RoboDK station: Raster Curve auto setup - Custom GUI.rdk

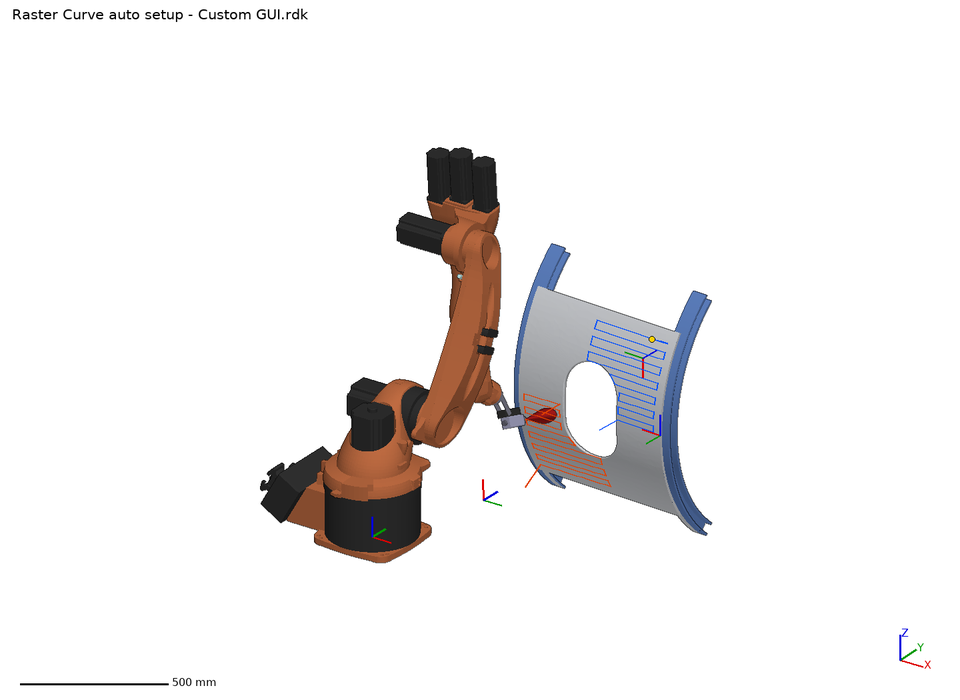
[picture v0: the station drawn from its stored meshes, robots at their saved joint values, targets as dots, program paths as lines]
Station Add curve sample project CreatePoint. Poses are relative to the parent item; angles as X-Y-Z fixed-axis rotations.
Station parameters (name, value as stored): IO_5, 0, CURVE_PARAMETERS, 600  600  250  250, STEP_X, 25.0, STEP_Y, 25.0, SPEED_OPERATION, 20.0, REPEAT_TIMES, 1.0, REPEAT_OFFSET, 2.0, ANGLE_TCP_X, 0.0, ANGLE_TCP_Y, -30.0, OVERTRAVEL, 25.0, SIZE_X, 300.0, SIZE_Y, 300.0
  - frame KUKA KR 5 arc Base at (0, 0, 0) mm
    - robot KUKA KR 5 arc: 6 axes, payload 5 kg, reach 1411 mm, repeatability 0.04 mm, weight 127 kg
        modified DH rows (alpha deg, a mm, theta deg, d mm): 0, 0, 0, 400; -90, 180, 0, 0; 0, 600, -90, 0; -90, 120, 0, 620; 90, 0, 0, 0; -90, 0, 180, 115
        joint limits [-155, -180, -15, -350, -130, -350] to [155, 65, 158, 350, 130, 350]; home [0, -90, 90, 0, 0, 0]; saved at [-90.662, -65.515, 150.914, 153.218, 47.362, 35.247]
      - tool Paint gun, TCP at (25, 0, 225) mm, rotated rx 0 ry 30 rz 0 deg, size 101.6 x 139.9 x 235.8 mm
    - frame CAD reference at (526.25, 941.36, 152.38) mm, rotated rx 0 ry 0 rz 177.82 deg
      - object Inspection Part at (0, 0, 0) mm, size 656 x 251.4 x 904.5 mm, 19 curves, geometry from Do something->PointOperations DOSOMETHING %ID%
      - frame Section1 at (31.6, 54.02, 303.28) mm, rotated rx 0 ry 90 rz -90 deg
        - object Section1 at (0, 0, 0) mm
      - frame Section2 at (569.12, 235.23, -318.39) mm, rotated rx 41.21 ry -87.7 rz 48.72 deg
        - object Section2 at (0, 0, 0) mm
  - Python program PointOperations (listed below)
  - Python program Curve_Auto_Setup (listed below)
  - machining project Section1: rotZ(0) | rotz(0) | onStart | onPathStart | onApproach | onPoint | onRetract | onFinish | Extruder(%1) | default | default | OutOnMov(%1) | OutOffMov(%1) | onPathFinish
  - program Section1 (141 instructions, listed below)
  - machining project Section2: rotZ(0) | onStart | onPathStart | onApproach | onPoint | onRetract | onFinish | Extruder(%1) | default | default | OutOnMov(%1) | OutOffMov(%1) | onPathFinish
  - program Section2 (141 instructions, listed below)
  - program MainInspection Part (2 instructions, listed below)
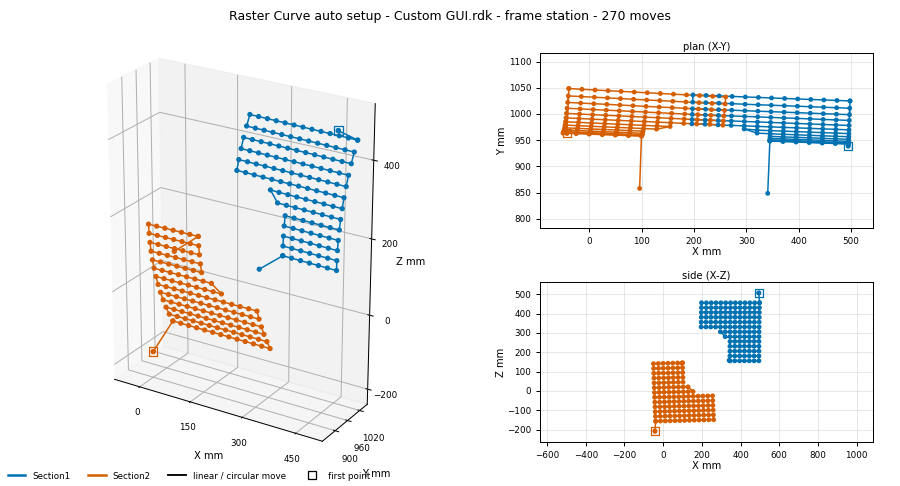
[picture p0: tool path of Raster Curve auto setup - Custom GUI.rdk in frame station, 270 of 270 moves have a stored position in this frame; points joined in program order, loops and branches not executed]

--- Python program PointOperations ---
import sys                # allows getting the argument parameters
from robodk import *      # required by mbox()
from robolink import *    # API to communicate with RoboDK

print('Number of arguments: ' + str(len(sys.argv)) + ' arguments.')

OBJECT = None
COMMAND = "SHOWPOINT_ALL"  # set to: NEWPOINT, SHOWPOINT

RDK = Robolink()

if len(sys.argv) >= 3:
    COMMAND = sys.argv[1]
    OBJECT = Item(RDK, int(sys.argv[2]))
    #RDK.ShowMessage("%s : %s" % (str(sys.argv), COMMAND))

else:
    OBJECT = RDK.ItemUserPick("Select an object", ITEM_TYPE_OBJECT)
    if not OBJECT.Valid():
        quit()

print("Selected object: %s" % OBJECT.Name())

if COMMAND == "SHOWPOINT_ALL":
    # Show all points in the object
    points, name = OBJECT.GetPoints(FEATURE_POINT)
    message = 'List of points for object<br>%s<br>' % OBJECT.Name()
    i = 0
    for pt in points:
        i = i + 1
        message += "p%i : %.3f , %.3f , %.3f <br>" % (i, pt[0], pt[1], pt[2])

    RDK.ShowMessage(message)

elif COMMAND == "SHOWPOINT":
    # Shows the point selected
    is_selected, feature_type, feature_id = OBJECT.SelectedFeature()
    points, name_selected = OBJECT.GetPoints(feature_type, feature_id)
    point = None
    if len(points) > 1:
        point = points[feature_id]
    else:
        point = points[0]
    RDK.ShowMessage("Selected Point: %s<br>XYZ = [%.3f, %.3f, %.3f]<br>ijk = [%.3f, %.3f, %.3f]" % (name_selected, point[0], point[1], point[2], point[3], point[4], point[5]))

elif COMMAND == "NEWPOINT":
    # create a new point under the mouse cursor
    point_mouse, name_feature = OBJECT.GetPoints(FEATURE_SURFACE)
    if 'point on surface' in name_feature.lower():
        point_rel = point_mouse[0]
        RDK.ShowMessage("%s -> XYZ = [%.3f, %.3f, %.3f] , ijk = [%.3f, %.3f, %.3f]" % (name_feature, point_rel[0], point_rel[1], point_rel[2], point_rel[3], point_rel[4], point_rel[5]), False)
        ADD_POINT_ON_OBJECT = True
        OBJECT.AddPoints([point_rel], ADD_POINT_ON_OBJECT, PROJECTION_NONE)
    else:
        RDK.ShowMessage("Select a surface")
else:
    raise Exception("Invalid operation specified")

--- Python program Curve_Auto_Setup ---
# Press F5 to run the script
# Type help("robolink") or help("robodk") for more information
#
# This script shows an example to create a raster curve that can be added programmatically to a RoboDK station
# The curve can be optionally projected to an existing object (either along the curve normals or a projection the closest surface)
#
# projection types (for AddCurve, as defined in robolink.py):
#PROJECTION_NONE                = 0 # No curve projection
#PROJECTION_CLOSEST             = 1 # The projection will the closest point on the surface
#PROJECTION_ALONG_NORMAL        = 2 # The projection will be done along the normal.
#PROJECTION_ALONG_NORMAL_RECALC = 3 # The projection will be done along the normal. Furthermore, the normal will be recalculated according to the surface normal.
#
# More information about the RoboDK API here:
# https://robodk.com/doc/en/PythonAPI/robolink.html
# https://robodk.com/doc/en/RoboDK-API.html
#
# This macro involves advanced Python programming as it uses the exec() and eval() statements to execute Python code from a string generated on the fly.
# The GUI is created automatically based on the variables defined in PARAM_VARS (global variables) and PARAM_LABELS (description to show on the menu)


# Set default/global parameters. This is only useful for the first time we execute this macro on a new RDK file.
# These global parameters are saved with the RoboDK station as Station parameters (right click the Station root and select "Station Parameters" to see the parameters saved)
SIZE_X = 500   # Size along the X axis
SIZE_Y = 500   # Size along the Y axis
STEP_X = 20    # Step along the X axis
STEP_Y = 50    # Step along the Y axis
SPEED_OPERATION = 20 # Operation speed
REPEAT_TIMES = 3    # Number of times to run the same program
REPEAT_OFFSET = 2   # Offset along Z axis in mm
ANGLE_TCP_X = 10
ANGLE_TCP_Y = 20
OVERTRAVEL = 25

REMEMBER_LAST_VALUES = True

#--------------------------------------------
# List the variables that will be remembered by the station and provided through the GUI
PARAM_VARS = []
PARAM_LABELS = []
PARAM_VARS += ["STEP_X", "STEP_Y"]
PARAM_LABELS += ["Step along X (mm)", "Step along Y (mm)"]

PARAM_VARS += ["SPEED_OPERATION"]
PARAM_LABELS +=  ["Operation speed (mm/s)"]

PARAM_VARS += ["REPEAT_TIMES", "REPEAT_OFFSET"]
PARAM_LABELS +=  ["Repeat times", "Repeat Offset along Z (mm)"]

PARAM_VARS += ["ANGLE_TCP_X", "ANGLE_TCP_Y"]
PARAM_LABELS +=  ["Tool angle X (deg)", "Tool angle Y (deg)"]

PARAM_VARS += ["OVERTRAVEL"]
PARAM_LABELS +=  ["Overtravel (mm)"]

PARAM_VARS += ["SIZE_X", "SIZE_Y"]
PARAM_LABELS += ["Size along X (mm)", "Size along Y (mm)"]

# Optionally provide a part name to auto select it without asking the user
PART_NAME = None # 'Paint Part'

#------------------------------------------------------------------
#--------------- PROGRAM START ---------------------
from robolink import *    # API to communicate with RoboDK
from robodk import *      # basic matrix operations

# Initialize the RoboDK API
RDK = Robolink()

# Set other constants:
TOL_PROJ_Z = sqrt(2)    # Tolerance to ignore a point as a ratio (if it falls through a window for example)

#---------------------------------------------
# First: Retrieve the part item
# Name of the reference used for the path projection
#

if PART_NAME is None:
    PART = RDK.ItemUserPick("Select a part", ITEM_TYPE_OBJECT)
    if PART is None:
        print("Operation cancelled by user")
        quit()
else:
    PART = RDK.Item(PART_NAME, ITEM_TYPE_OBJECT)

if not PART.Valid():
    raise Exception("The selected part is not valid or not available")

#---------------------------------------------
# List all the reference frames that we want to use to create
# raster paths (references attached to the object reference
part_ref = PART.Parent()

# Get the list of items attached to the part reference
ref_pattern_candidates = part_ref.Childs()
# Iterate through these child items and list the reference frames
# optionally add ignore in the name
REF_PATTERN_LIST = []
for ref_i in ref_pattern_candidates:
    if ref_i.Type() == ITEM_TYPE_FRAME and (not "ignore" in ref_i.Name()):
        REF_PATTERN_LIST.append(ref_i)

if len(REF_PATTERN_LIST) <= 0:
    RDK.ShowMessage("No reference frames found. Add one or more frames to " + part_ref.Name())
    quit()

#---------------------------------------------
# Retrieve Global parameters or set defaults as found in RoboDK
if REMEMBER_LAST_VALUES:
    for strvar in PARAM_VARS:
        var_value = RDK.getParam(strvar)
        if var_value is not None:
            exec(strvar + " = " + str(var_value))

#---------------------------------------------
# Load GUI tools
from tkinter import *
import tkinter.font as font

# Generate the main window
root = Tk()
root.title("Toolpath parameters")

# define a label to notify the user
NotifyGUI = StringVar()

#---------------------------------------------
# Function to change the coordinates of a point and a normal
# given a pose. The point and the normal must be in xyzijk format
def Pose_x_XYZijk(pose, xyzijk):
    new_xyz = pose*xyzijk[0:3]
    new_ijk = pose[:3,:3]*xyzijk[3:6]
    return new_xyz + new_ijk

#---------------------------------------------
# Function definition to create a list of points as zig-zag pattern (curve)
def GridPoints(ref, size_x, size_y, step_x, step_y):
    """Generates a list of points given dimensions of a grid"""
    points = []
    xx = 0
    flip = 1
    while xx <= size_x:
        yy = 0
        if flip > 0:
            yy = 0
        else:
            yy = size_y

        while yy <= size_y and yy >= 0:
            # Create a new point as [x,y,z , i,j,k]
            xyzijk = Pose_x_XYZijk(ref, [xx,yy,0 , 0,0,-1])
            points.append(xyzijk)
            yy = yy + flip*step_y

        xx = xx + step_x
        flip = -1*flip
    return points

#---------------------------------------------
# Function definition to offset a list of points
def PointsOffset(points, offset):
    points_offset = []
    for pi in points:
        x,y,z,i,j,k = pi
        xyz2 = add3([x,y,z], mult3([i,j,k], offset))
        xyzijk2 = xyz2 + [i,j,k]
        points_offset.append(xyzijk2)
    return points_offset

# Show message through the GUI, RoboDK and the console
def ShowMsg(msg):
    print(msg)
    NotifyGUI.set(msg)
    root.update_idletasks()
    RDK.ShowMessage(msg, False)

#---------------------------------------------
# Main program call that will project the path to a surface
def CreatePaths():
    prog_name_list = []
    for REF in REF_PATTERN_LIST:
        # Retrieve the reference name
        REF_NAME = REF.Name()

        ShowMsg("Working with %s ..." % REF_NAME)

        # Get the pose of the reference with respect to the part:
        pose_ref_wrt_part = invH(PART.Parent().PoseAbs())*REF.PoseAbs()

        # For later: calculate the inverse pose (part with respect to the reference)
        pose_part_wrt_ref = invH(pose_ref_wrt_part)

        # Generate the curve path
        # IMPORTANT: the point coordinates must be relative to the part reference
        points = GridPoints(pose_ref_wrt_part, SIZE_X, SIZE_Y, STEP_X, STEP_Y)
        # points is a list of points with respect to the part
        # Another option is to load the grid from a CSV file:
        #file = RDK.getParam('PATH_OPENSTATION') + '/test.csv'
        #POINTS = LoadList(file)
        #POINTS.pop(0)
        # display the points
        #print(CURVE)
        if len(points) == 0:
            ShowMsg("No points found for: " + REF_NAME)
            continue

        # Project the points on the object surface
        #pts_projected = PART.AddPoints(POINTS)
        ShowMsg("Projecting %s to surface..." % REF_NAME)
        points_projected = PART.ProjectPoints(Mat(points).tr(), PROJECTION_ALONG_NORMAL_RECALC)

        # Patch
        points_projected = points_projected.tr().rows

        points_projected_filtered = []

        ShowMsg("Filtering %s..." % REF_NAME)

        # Remember the last valid projection
        pti_last = None
        for i in range(0,len(points_projected)-1):
            # retrieve projected and non projected points, with respect to the reference frame
            # retrieve the next point to test if the projection went too far
            pti = Pose_x_XYZijk(pose_part_wrt_ref, points[i])
            pti_proj = Pose_x_XYZijk(pose_part_wrt_ref, points_projected[i])

            # Ignore non projected points (z coordinate is 0 mm, prevent numerical errors as well)
            if abs(pti_proj[2]) < 0.1:
                continue

            # Check if we have the first valid projected point
            if pti_last is None:
                points_projected_filtered.append(pti_proj)
                pti_last = pti
                pti_proj_last = pti_proj
                continue

            # Check if the projection falls through a "window" or "climbs" a wall with respect to the previous pointS
            if distance(pti_proj, pti_proj_last) < TOL_PROJ_Z*distance(pti, pti_last):
                # List the point as valid
                points_projected_filtered.append(pti_proj)

                # Remember the last valid projection
                pti_last = pti
                pti_proj_last = pti_proj

        # Remove any previously generated objects with the same name as the reference frame:
        obj_delete = RDK.Item(REF_NAME, ITEM_TYPE_OBJECT)
        if obj_delete.Valid():
            obj_delete.Delete()

        ShowMsg("Creating object for %s..." % REF_NAME)
        # Add the points as an object in the RoboDK station tree
        points_object = RDK.AddCurve(points_projected_filtered)
        # Add the points to the reference and set the reference name
        points_object.setParent(REF)
        points_object.setName(REF_NAME)

        for rep in range(1,round(REPEAT_TIMES)):
            # Calculate a new curve with respect to the reference curve
            points_projected_filtered_rep = PointsOffset(points_projected_filtered, REPEAT_OFFSET * rep)

            #  Add the shifted curve without projecting it
            points_object = RDK.AddCurve(points_projected_filtered_rep, points_object, True, PROJECTION_NONE)


        curve_follow = RDK.Item(REF_NAME, ITEM_TYPE_MACHINING)
        if not curve_follow.Valid():
            curve_follow = RDK.AddMillingProject(REF_NAME)

        ShowMsg("Solving toolpath for %s" % REF_NAME)

        # Use the current reference frame:
        curve_follow.setPoseFrame(REF)

        # RoboDK 3.3.7 or later required:
        curve_follow.setSpeed(SPEED_OPERATION)
        curve_follow.setPoseTool(rotx(ANGLE_TCP_X*pi/180.0)*roty(ANGLE_TCP_Y*pi/180.0))
        prog, status = curve_follow.setMillingParameters(part=points_object)
        print(status)
        if status == 0:
            ShowMsg("Program %s generated successfully" % REF_NAME)
        else:
            ShowMsg("Issues found generating program %s!" % REF_NAME)


        # get the program name
        prog_name = prog.Name()
        prog_name_list.append(prog_name)

    # Create a new program that calls the auto generated program
    # Make sure we delete any previously generated programs with the same name
    ShowMsg("Creating Main program ...")
    prog_main_name = "Main" + PART.Name()
    prog_main = RDK.Item(prog_main_name, ITEM_TYPE_PROGRAM)
    if prog_main.Valid():
        prog_main.Delete()
    prog_main = RDK.AddProgram(prog_main_name)

    # Add a number of program calls to the first program by providing inline code
    #prog_main.RunCodeCustom("FOR i=1 TO 5", INSTRUCTION_INSERT_CODE)
    #prog_main.RunCodeCustom(prog_name, INSTRUCTION_CALL_PROGRAM)
    #prog_main.RunCodeCustom("NEXT", INSTRUCTION_INSERT_CODE)
    #for i in range(4):
    for pr_name in prog_name_list:
        prog_main.RunCodeCustom(pr_name, INSTRUCTION_CALL_PROGRAM)


    # Start the program simulation:
    prog_main.RunProgram()
    ShowMsg("Done!!")


#-----------------------------------------
# Create a GUI menu using tkinter



# Use StringVar variables linked to the global variables for the GUI
txtSpeed_Operation = StringVar()
txtSpeed_Operation.set(str(SPEED_OPERATION))


for strvar, hint in zip(PARAM_VARS, PARAM_LABELS):
    var = eval(strvar)
    txtvar = "txt" + strvar
    #txtSize_X = StringVar()
    #txtSize_X.set(str(SIZE_X))
    #Label(root, text="Window Size X (mm)").pack()
    #Entry(root, textvariable=txtSize_X).pack()
    exec(txtvar + " = StringVar()")
    exec(txtvar + ".set(str(" + str(var) + "))")
    exec("Label(root, text='" + hint + "').pack()")
    exec("Entry(root, textvariable=" + txtvar + ").pack()")


# Add a button and default action to execute the current choice of the user
def btnUpdate():
    # List the global variables so that we can read or modify the latest values
    #exec(PARAM_GLOBALS)

    try:
        for strvar in PARAM_VARS:
            #SIZE_X = float(txtSize_X.get())
            # Update global variable
            exec("%s = float(txt%s.get())" % (strvar, strvar), globals())

    except Exception as e:
        RDK.ShowMessage("Invalid input!! " + str(e), False)
        return

    # Remember the last settings in the RoboDK station
    for strvar in PARAM_VARS:
        value = eval(strvar)
        RDK.setParam(strvar, value)

    # Run the main program once all the global variables have been set
    CreatePaths()

# Add an update button that calls btnUpdate()
font_large = font.Font(family='Helvetica', size=18, weight=font.BOLD)
Label(root, text=" ").pack() # Just a spacer
Label(root, textvariable=NotifyGUI).pack() # information variable
Button(root, text='Update', font=font_large, width=20, height=4, command=btnUpdate, bg='green').pack()

# Important to display the graphical user interface
root.mainloop()

--- program Section1 (robot KUKA KR 5 arc) ---
  Set Ref.: Section1
  Set Tool: Paint gun
  Show Paint gun
  Set speed (1000.0 mm/s)
  MoveJ 1 to (-50.79, 0.22, 50.26) mm, rotated rx 34.39 ry 25.95 rz 105.39 deg; joints [-51.825, -81.117, 121.806, -97.903, 30.623, 30.499]
  MoveL 2 to (-50.79, 0.22, 50.26) mm, rotated rx 34.39 ry 25.95 rz 105.39 deg; joints [-51.825, -81.117, 121.806, -97.903, 30.623, 30.499]
  MoveL 3 to (0, 0, 136.4) mm, rotated rx 34.39 ry 25.95 rz 105.39 deg; joints [-55.067, -72.344, 116.19, -106.364, 28.938, 37.73]
  MoveL 4 to (0, 0, 136.4) mm, rotated rx 34.39 ry 25.95 rz 105.39 deg; joints [-55.067, -72.344, 116.19, -106.364, 28.938, 37.73]
  Set speed (20.0 mm/s)
  MoveL 5 to (0, 25, 136.39) mm, rotated rx 34.36 ry 26.11 rz 105.47 deg; joints [-56.374, -73.392, 117.629, -108.355, 28.338, 38.991]
  MoveL 6 to (0, 50, 136.37) mm, rotated rx 34.57 ry 26.16 rz 105.61 deg; joints [-57.765, -74.441, 118.921, -109.961, 27.461, 39.815]
  MoveL 7 to (0, 75, 136.32) mm, rotated rx 34.08 ry 26.14 rz 105.33 deg; joints [-59.224, -75.485, 120.503, -113.62, 26.851, 42.548]
  MoveL 8 to (0, 100, 136.36) mm, rotated rx 35.34 ry 25.72 rz 105.77 deg; joints [-60.883, -76.578, 121.224, -113.176, 24.731, 41.191]
  MoveL 9 to (0, 125, 136.35) mm, rotated rx 34.79 ry 26.08 rz 105.68 deg; joints [-62.268, -77.415, 122.604, -116.74, 24.649, 43.9]
  MoveL 10 to (0, 150, 136.37) mm, rotated rx 33.98 ry 26.51 rz 105.48 deg; joints [-63.673, -78.184, 124.024, -120.948, 24.856, 47.226]
  MoveL 11 to (0, 175, 136.42) mm, rotated rx 34.8 ry 25.76 rz 105.5 deg; joints [-65.595, -79.234, 124.78, -122.936, 22.472, 48.001]
  MoveL 12 to (0, 200, 136.37) mm, rotated rx 35.19 ry 25.98 rz 105.85 deg; joints [-67.131, -79.96, 125.512, -124.323, 21.617, 48.504]
  MoveL 13 to (0, 225, 136.46) mm, rotated rx 34.52 ry 25.87 rz 105.41 deg; joints [-68.896, -80.721, 126.726, -130.032, 21.139, 53.027]
  MoveL 14 to (0, 250, 136.49) mm, rotated rx 34.38 ry 26.44 rz 105.66 deg; joints [-70.36, -81.256, 127.529, -132.471, 21.131, 54.622]
  MoveL 15 to (0, 275, 136.38) mm, rotated rx 34.16 ry 25.74 rz 105.14 deg; joints [-72.462, -82.045, 128.43, -139.005, 19.726, 59.712]
  MoveL 16 to (0, 300, 136.48) mm, rotated rx 34.45 ry 26.26 rz 105.6 deg; joints [-73.982, -82.481, 128.889, -140.551, 19.313, 60.407]
  MoveL 17 to (25, 300, 122.63) mm, rotated rx 31.54 ry 26.48 rz 104.15 deg; joints [-73.798, -81.794, 132.47, -150.222, 25.031, 70.279]
  MoveL 18 to (25, 275, 122.58) mm, rotated rx 31.34 ry 26.67 rz 104.15 deg; joints [-71.878, -81.182, 131.886, -146.426, 25.961, 67.747]
  MoveL 19 to (25, 250, 122.59) mm, rotated rx 31.37 ry 26.79 rz 104.22 deg; joints [-70.021, -80.535, 131.115, -142.618, 26.6, 65.164]
  MoveL 20 to (25, 225, 122.63) mm, rotated rx 31.4 ry 26.19 rz 103.93 deg; joints [-68.532, -80.013, 130.364, -140.83, 26.566, 64.202]
  MoveL 21 to (25, 200, 122.46) mm, rotated rx 31.14 ry 26.76 rz 104.09 deg; joints [-66.547, -79.122, 129.511, -136.799, 28.011, 61.538]
  MoveL 22 to (25, 175, 122.46) mm, rotated rx 31.13 ry 26.9 rz 104.15 deg; joints [-64.795, -78.29, 128.512, -133.535, 28.801, 59.418]
  MoveL 23 to (25, 150, 122.52) mm, rotated rx 31.21 ry 27.02 rz 104.25 deg; joints [-63.098, -77.413, 127.39, -130.303, 29.498, 57.291]
  MoveL 24 to (25, 125, 122.54) mm, rotated rx 30.85 ry 26.24 rz 103.67 deg; joints [-61.827, -76.744, 126.591, -129.936, 29.622, 57.505]
  MoveL 25 to (25, 100, 122.49) mm, rotated rx 30.04 ry 26.97 rz 103.61 deg; joints [-59.962, -75.527, 125.569, -127.468, 31.746, 56.269]
  MoveL 26 to (25, 75, 122.47) mm, rotated rx 30.04 ry 26.97 rz 103.61 deg; joints [-58.439, -74.554, 124.29, -124.982, 32.356, 54.711]
  MoveL 27 to (25, 50, 122.46) mm, rotated rx 31.64 ry 26.69 rz 104.31 deg; joints [-57.078, -73.733, 122.317, -119.835, 31.394, 50.498]
  MoveL 28 to (25, 25, 122.49) mm, rotated rx 30.53 ry 27.39 rz 104.08 deg; joints [-55.375, -72.363, 121.164, -118.632, 33.673, 50.336]
  MoveL 29 to (25, 0, 122.49) mm, rotated rx 30.01 ry 27 rz 103.61 deg; joints [-54.125, -71.378, 120.016, -118.051, 34.238, 50.323]
  MoveL 30 to (50, 0, 110.15) mm, rotated rx 27.7 ry 28.02 rz 102.88 deg; joints [-53.265, -69.968, 122.392, -122.88, 38.773, 56.45]
  MoveL 31 to (50, 25, 110.15) mm, rotated rx 28.68 ry 27.24 rz 103.03 deg; joints [-54.96, -71.439, 123.802, -124.84, 36.682, 57.29]
  MoveL 32 to (50, 50, 110.13) mm, rotated rx 27.17 ry 27.18 rz 102.23 deg; joints [-56.415, -72.299, 125.849, -129.594, 37.607, 60.996]
  MoveL 33 to (50, 75, 110.14) mm, rotated rx 28.79 ry 27.09 rz 103.02 deg; joints [-57.961, -73.539, 126.619, -129.604, 35.483, 60.198]
  MoveL 34 to (50, 100, 110.18) mm, rotated rx 28.44 ry 26.87 rz 102.73 deg; joints [-59.593, -74.521, 128.109, -133.043, 35.156, 62.519]
  MoveL 35 to (50, 125, 110.18) mm, rotated rx 27.77 ry 27.25 rz 102.56 deg; joints [-61.029, -75.217, 129.49, -135.829, 35.745, 64.444]
  MoveL 36 to (50, 150, 110.13) mm, rotated rx 27.07 ry 27.33 rz 102.24 deg; joints [-62.635, -75.952, 130.892, -139.242, 36.153, 66.789]
  MoveL 37 to (50, 175, 110.15) mm, rotated rx 28.38 ry 27.14 rz 102.83 deg; joints [-64.383, -77.036, 131.506, -140.401, 34.089, 66.885]
  MoveL 38 to (50, 200, 110.12) mm, rotated rx 27.77 ry 27.52 rz 102.69 deg; joints [-65.947, -77.606, 132.664, -143.206, 34.669, 68.73]
  MoveL 39 to (50, 225, 110.16) mm, rotated rx 28.95 ry 27.22 rz 103.17 deg; joints [-67.817, -78.596, 133.181, -145.031, 32.612, 69.343]
  MoveL 40 to (50, 250, 110.12) mm, rotated rx 29.34 ry 27.22 rz 103.36 deg; joints [-69.606, -79.328, 133.876, -147.475, 31.723, 70.637]
  MoveL 41 to (50, 275, 110.11) mm, rotated rx 29.3 ry 27.08 rz 103.27 deg; joints [-71.512, -79.974, 134.671, -150.994, 31.233, 72.848]
  MoveL 42 to (50, 300, 110.16) mm, rotated rx 28.95 ry 27.21 rz 103.16 deg; joints [-73.336, -80.434, 135.461, -154.319, 31.387, 74.966]
  MoveL 43 to (75, 300, 99.17) mm, rotated rx 26.35 ry 27.87 rz 102.11 deg; joints [-72.914, -78.494, 138.029, -157.061, 37.959, 78.371]
  MoveL 44 to (75, 275, 99.15) mm, rotated rx 24.89 ry 28.03 rz 101.43 deg; joints [-70.979, -77.558, 137.792, -155.248, 40.23, 77.838]
  MoveL 45 to (75, 250, 99.18) mm, rotated rx 26.18 ry 28.52 rz 102.29 deg; joints [-68.83, -77.135, 136.49, -150.194, 39.161, 74.534]
  MoveL 46 to (75, 225, 99.19) mm, rotated rx 24.45 ry 28.23 rz 101.29 deg; joints [-67.174, -76.147, 136.24, -149.877, 41.421, 75.117]
  MoveL 47 to (75, 200, 99.17) mm, rotated rx 26.06 ry 27.88 rz 101.96 deg; joints [-65.506, -75.928, 134.84, -146.333, 39.442, 72.689]
  MoveL 48 to (75, 175, 99.35) mm, rotated rx 25.32 ry 27.81 rz 101.56 deg; joints [-63.803, -75.016, 134.065, -144.716, 40.579, 72.132]
  MoveL 49 to (75, 150, 99.2) mm, rotated rx 24.89 ry 27.44 rz 101.19 deg; joints [-62.255, -74.246, 133.218, -143.422, 41.114, 71.694]
  MoveL 50 to (75, 125, 99.26) mm, rotated rx 25.57 ry 28.07 rz 101.79 deg; joints [-60.332, -73.353, 131.644, -139.022, 41.053, 68.839]
  MoveL 51 to (75, 100, 99.29) mm, rotated rx 25.97 ry 27.78 rz 101.88 deg; joints [-58.843, -72.636, 130.337, -136.714, 40.684, 67.42]
  MoveL 52 to (75, 75, 99.2) mm, rotated rx 25.28 ry 27.8 rz 101.53 deg; joints [-57.272, -71.572, 129.254, -135.206, 41.76, 66.857]
  MoveL 53 to (75, 50, 99.17) mm, rotated rx 26.54 ry 27.82 rz 102.19 deg; joints [-55.763, -70.839, 127.419, -131.31, 40.727, 64.018]
  MoveL 54 to (75, 25, 99.18) mm, rotated rx 24.66 ry 28.53 rz 101.51 deg; joints [-54.02, -69.23, 126.337, -130.26, 43.556, 64.121]
  MoveL 55 to (75, 0, 99.19) mm, rotated rx 26.41 ry 27.32 rz 101.9 deg; joints [-53.07, -68.946, 124.647, -127.962, 41.071, 62.108]
  MoveL 56 to (100, 0, 89.53) mm, rotated rx 23.57 ry 27.8 rz 100.68 deg; joints [-52.461, -66.851, 126.641, -132.117, 46.26, 67.396]
  MoveL 57 to (100, 25, 89.51) mm, rotated rx 21.6 ry 29.11 rz 100.17 deg; joints [-53.388, -66.892, 128.248, -133.924, 49.194, 69.081]
  MoveL 58 to (100, 50, 89.53) mm, rotated rx 22.91 ry 28.2 rz 100.5 deg; joints [-55.21, -68.499, 129.717, -136.304, 47.004, 70.032]
  MoveL 59 to (100, 75, 89.52) mm, rotated rx 22.45 ry 28.42 rz 100.35 deg; joints [-56.649, -69.223, 131.187, -138.51, 47.555, 71.396]
  MoveL 60 to (100, 100, 89.57) mm, rotated rx 23.15 ry 27.97 rz 100.53 deg; joints [-58.408, -70.438, 132.473, -140.848, 46.308, 72.451]
  MoveL 61 to (100, 125, 89.57) mm, rotated rx 23.38 ry 28.52 rz 100.85 deg; joints [-59.812, -71.173, 133.509, -141.91, 46.235, 72.835]
  MoveL 62 to (100, 150, 89.59) mm, rotated rx 23.03 ry 28.17 rz 100.55 deg; joints [-61.636, -71.992, 134.906, -145.168, 46.3, 74.696]
  MoveL 63 to (100, 175, 89.57) mm, rotated rx 22.81 ry 28.32 rz 100.49 deg; joints [-63.3, -72.641, 136.048, -147.424, 46.539, 75.87]
  MoveL 64 to (100, 200, 89.57) mm, rotated rx 22.58 ry 28.26 rz 100.36 deg; joints [-65.104, -73.303, 137.166, -150.099, 46.669, 77.261]
  MoveL 65 to (100, 225, 89.57) mm, rotated rx 22.42 ry 28.41 rz 100.33 deg; joints [-66.864, -73.876, 138.138, -152.375, 46.842, 78.361]
  MoveL 66 to (100, 250, 89.52) mm, rotated rx 23.05 ry 28.39 rz 100.64 deg; joints [-68.73, -74.704, 138.857, -154.444, 45.856, 79.138]
  MoveL 67 to (100, 275, 89.52) mm, rotated rx 21.87 ry 28.55 rz 100.11 deg; joints [-70.598, -74.838, 139.945, -157.482, 47.427, 80.844]
  MoveL 68 to (100, 300, 89.53) mm, rotated rx 22.58 ry 28.21 rz 100.34 deg; joints [-72.693, -75.665, 140.525, -160.252, 46.175, 82.002]
  MoveL 69 to (125, 300, 81.15) mm, rotated rx 20.36 ry 28.41 rz 99.31 deg; joints [-72.485, -72.746, 142.125, -161.759, 52.405, 84.09]
  MoveL 70 to (125, 275, 81.51) mm, rotated rx -9.72 ry 31.15 rz 85.26 deg; joints [-69.41, -54.992, 140.943, -160.257, 94.501, 88.519]
  MoveL 71 to (125, 250, 81.14) mm, rotated rx 13.43 ry 28.51 rz 96.05 deg; joints [-68.612, -68.639, 141.777, -159.707, 62.306, 84.736]
  MoveL 72 to (125, 225, 81.15) mm, rotated rx 20.42 ry 28.31 rz 99.31 deg; joints [-66.701, -71.242, 139.721, -154.724, 52.26, 81.3]
  MoveL 73 to (125, 200, 81.17) mm, rotated rx 19.09 ry 28.99 rz 98.87 deg; joints [-64.561, -69.93, 138.858, -151.99, 54.338, 80.415]
  MoveL 74 to (125, 175, 81.15) mm, rotated rx 19.63 ry 28.62 rz 99.02 deg; joints [-62.914, -69.582, 137.787, -150.069, 53.427, 79.497]
  MoveL 75 to (125, 150, 81.14) mm, rotated rx 19.39 ry 28.96 rz 99.01 deg; joints [-61.02, -68.698, 136.601, -147.424, 53.852, 78.348]
  MoveL 76 to (125, 125, 81.16) mm, rotated rx 19.1 ry 29.06 rz 98.9 deg; joints [-59.284, -67.819, 135.409, -145.291, 54.229, 77.447]
  MoveL 77 to (125, 100, 81.16) mm, rotated rx 19.44 ry 28.9 rz 99.01 deg; joints [-57.708, -67.207, 134.102, -143.242, 53.686, 76.379]
  MoveL 78 to (125, 75, 81.13) mm, rotated rx 20.02 ry 28.69 rz 99.24 deg; joints [-56.199, -66.648, 132.687, -141.099, 52.83, 75.141]
  MoveL 79 to (125, 50, 81.14) mm, rotated rx 20.03 ry 28.69 rz 99.24 deg; joints [-54.662, -65.793, 131.253, -139.048, 52.78, 74.067]
  MoveL 80 to (125, 25, 81.13) mm, rotated rx 20.01 ry 28.64 rz 99.22 deg; joints [-53.191, -64.906, 129.773, -137.124, 52.745, 73.029]
  MoveL 81 to (125, 0, 81.13) mm, rotated rx 18.59 ry 28.92 rz 98.61 deg; joints [-51.632, -63.439, 128.389, -135.763, 54.5, 72.674]
  MoveL 82 to (150, 0, 73.98) mm, rotated rx 15.95 ry 28.88 rz 97.32 deg; joints [-51.3, -60.627, 129.519, -138.302, 59.576, 76.307]
  MoveL 83 to (150, 25, 73.95) mm, rotated rx 18.14 ry 29.36 rz 98.51 deg; joints [-52.617, -62.151, 130.564, -138.167, 57.312, 75.692]
  MoveL 84 to (150, 50, 73.94) mm, rotated rx 17.05 ry 29.07 rz 97.9 deg; joints [-54.195, -62.66, 132.375, -141.181, 58.711, 77.558]
  MoveL 85 to (150, 75, 73.94) mm, rotated rx 16.37 ry 29.17 rz 97.59 deg; joints [-55.699, -63.142, 133.885, -143.33, 59.81, 78.797]
  MoveL 86 to (150, 100, 73.95) mm, rotated rx 17.08 ry 29.11 rz 97.93 deg; joints [-57.332, -64.195, 135.171, -145.037, 59.076, 79.395]
  MoveL 87 to (150, 125, 73.96) mm, rotated rx 16.61 ry 28.99 rz 97.67 deg; joints [-59.037, -64.741, 136.582, -147.49, 59.846, 80.608]
  MoveL 88 to (150, 150, 73.94) mm, rotated rx 17.03 ry 28.95 rz 97.85 deg; joints [-60.773, -65.604, 137.76, -149.435, 59.472, 81.308]
  MoveL 89 to (150, 175, 73.97) mm, rotated rx 17.54 ry 28.68 rz 98.03 deg; joints [-62.655, -66.527, 138.899, -151.744, 58.872, 82.112]
  MoveL 90 to (150, 200, 75.26) mm, rotated rx -26.35 ry 2.51 rz 89.84 deg; joints [-77.888, -41.231, 134.902, -200.878, 116.123, 74.828]
  MoveL 91 to (175, 175, 68.25) mm, rotated rx -0.98 ry 10.78 rz 89.85 deg; joints [-71.001, -54.636, 142.105, -182.397, 88.364, 89.756]
  MoveL 92 to (175, 150, 67.97) mm, rotated rx 14.13 ry 29.15 rz 96.52 deg; joints [-60.468, -61.82, 138.468, -150.76, 65.911, 83.877]
  MoveL 93 to (175, 125, 67.92) mm, rotated rx 14.96 ry 29.35 rz 96.96 deg; joints [-58.659, -61.579, 137.099, -148.159, 64.501, 82.688]
  MoveL 94 to (175, 100, 67.9) mm, rotated rx 13.88 ry 29.39 rz 96.45 deg; joints [-56.966, -60.434, 135.882, -146.555, 65.595, 82.31]
  MoveL 95 to (175, 75, 67.9) mm, rotated rx 13.88 ry 29.38 rz 96.44 deg; joints [-55.355, -59.774, 134.507, -144.67, 65.24, 81.495]
  MoveL 96 to (175, 50, 67.9) mm, rotated rx 13.67 ry 29.43 rz 96.36 deg; joints [-53.772, -58.969, 133.052, -142.798, 65.157, 80.682]
  MoveL 97 to (175, 25, 67.95) mm, rotated rx 13.16 ry 29.52 rz 96.13 deg; joints [-52.234, -57.995, 131.536, -141.059, 65.44, 79.946]
  MoveL 98 to (175, 0, 67.96) mm, rotated rx 13.44 ry 29.22 rz 96.2 deg; joints [-50.886, -57.431, 130.047, -139.594, 64.661, 79.074]
  MoveL 99 to (200, 0, 63) mm, rotated rx 10.52 ry 29.33 rz 94.85 deg; joints [-50.594, -53.847, 130.275, -140.913, 70.125, 81.778]
  MoveL 100 to (200, 25, 63.01) mm, rotated rx 10.87 ry 29.74 rz 95.08 deg; joints [-51.917, -54.588, 131.679, -141.928, 70.254, 82.307]
  MoveL 101 to (200, 50, 63.04) mm, rotated rx 11.35 ry 29.65 rz 95.3 deg; joints [-53.464, -55.481, 133.221, -143.672, 70.139, 83.024]
  MoveL 102 to (200, 75, 63.05) mm, rotated rx 11.69 ry 29.21 rz 95.38 deg; joints [-55.198, -56.355, 134.827, -146.027, 70.148, 83.932]
  MoveL 103 to (200, 100, 63.08) mm, rotated rx 12.13 ry 29.92 rz 95.72 deg; joints [-56.56, -56.995, 135.928, -146.708, 70.157, 84.17]
  MoveL 104 to (200, 125, 62.98) mm, rotated rx 11.56 ry 29.62 rz 95.39 deg; joints [-58.344, -57.317, 137.368, -149.173, 71.359, 85.209]
  MoveL 105 to (200, 150, 63.02) mm, rotated rx 12.2 ry 29.68 rz 95.7 deg; joints [-60.065, -58.143, 138.562, -150.86, 70.997, 85.639]
  MoveL 106 to (225, 150, 59.17) mm, rotated rx 8.57 ry 29.93 rz 94.02 deg; joints [-59.81, -53.39, 138.314, -151.406, 78.115, 87.812]
  MoveL 107 to (225, 125, 59.22) mm, rotated rx 9.31 ry 30.2 rz 94.41 deg; joints [-57.96, -53.341, 137.014, -149.029, 76.512, 86.952]
  MoveL 108 to (225, 100, 59.17) mm, rotated rx 9.42 ry 29.67 rz 94.38 deg; joints [-56.476, -53.042, 135.906, -147.943, 75.748, 86.495]
  MoveL 109 to (225, 75, 59.15) mm, rotated rx 9.54 ry 29.67 rz 94.44 deg; joints [-54.848, -52.613, 134.54, -146.141, 74.981, 85.783]
  MoveL 110 to (225, 50, 59.15) mm, rotated rx 7.83 ry 29.78 rz 93.65 deg; joints [-53.22, -51.189, 132.994, -144.568, 76.494, 85.485]
  MoveL 111 to (225, 25, 59.16) mm, rotated rx 9.49 ry 29.72 rz 94.42 deg; joints [-51.742, -51.487, 131.56, -142.613, 73.808, 84.238]
  MoveL 112 to (225, 0, 59.15) mm, rotated rx 8.24 ry 29.8 rz 93.85 deg; joints [-50.243, -50.265, 129.911, -141.121, 74.711, 83.739]
  MoveL 113 to (250, 0, 56.4) mm, rotated rx 5.71 ry 29.7 rz 92.65 deg; joints [-50.128, -46.527, 129.389, -141.896, 79.397, 85.79]
  MoveL 114 to (250, 25, 56.45) mm, rotated rx 5.68 ry 29.97 rz 92.66 deg; joints [-51.506, -46.965, 130.842, -143.136, 80.163, 86.498]
  MoveL 115 to (250, 50, 56.47) mm, rotated rx 7.1 ry 29.56 rz 93.28 deg; joints [-53.178, -48.242, 132.627, -145.157, 79.211, 87.041]
  MoveL 116 to (250, 75, 56.46) mm, rotated rx 7.13 ry 30.12 rz 93.36 deg; joints [-54.554, -48.612, 133.848, -146.063, 79.873, 87.53]
  MoveL 117 to (250, 100, 56.54) mm, rotated rx 5.61 ry 29.68 rz 92.6 deg; joints [-56.347, -48.228, 135.222, -148.571, 82.56, 88.631]
  MoveL 118 to (250, 125, 56.46) mm, rotated rx 5.28 ry 30.08 rz 92.48 deg; joints [-57.883, -48.335, 136.336, -149.786, 83.705, 89.15]
  MoveL 119 to (250, 150, 56.51) mm, rotated rx 6.04 ry 30.16 rz 92.84 deg; joints [-59.608, -49.077, 137.602, -151.43, 83.487, 89.464]
  MoveL 120 to (275, 150, 54.74) mm, rotated rx 3.6 ry 29.56 rz 91.66 deg; joints [-59.781, -44.829, 136.772, -152.386, 88.591, 91.042]
  MoveL 121 to (275, 125, 54.7) mm, rotated rx 3.3 ry 30.02 rz 91.54 deg; joints [-57.834, -44.382, 135.388, -149.976, 88.013, 90.61]
  MoveL 122 to (275, 100, 54.76) mm, rotated rx 3.41 ry 30.21 rz 91.6 deg; joints [-56.067, -44.156, 134.063, -147.994, 86.977, 90.05]
  MoveL 123 to (275, 75, 54.71) mm, rotated rx 2.64 ry 30.04 rz 91.23 deg; joints [-54.488, -43.438, 132.66, -146.58, 87.069, 89.655]
  MoveL 124 to (275, 50, 54.71) mm, rotated rx 2.63 ry 29.91 rz 91.23 deg; joints [-52.955, -43.117, 131.295, -145.141, 86.225, 89.048]
  MoveL 125 to (275, 25, 54.73) mm, rotated rx 3.65 ry 30.04 rz 91.71 deg; joints [-51.394, -43.281, 129.916, -143.326, 84.136, 88.103]
  MoveL 126 to (275, 0, 54.7) mm, rotated rx 3.08 ry 29.97 rz 91.44 deg; joints [-49.952, -42.57, 128.31, -141.931, 83.973, 87.473]
  MoveL 127 to (300, 0, 54.07) mm, rotated rx 0.88 ry 30 rz 90.41 deg; joints [-49.907, -38.819, 127.024, -142.055, 87.824, 88.925]
  MoveL 128 to (300, 25, 54.07) mm, rotated rx 0.88 ry 30 rz 90.41 deg; joints [-51.372, -39.159, 128.559, -143.542, 88.757, 89.672]
  MoveL 129 to (300, 50, 54.07) mm, rotated rx 0.88 ry 30 rz 90.41 deg; joints [-52.894, -39.46, 130.024, -145.073, 89.701, 90.351]
  MoveL 130 to (300, 75, 54.07) mm, rotated rx 0.88 ry 30 rz 90.41 deg; joints [-54.474, -39.724, 131.417, -146.651, 90.654, 90.96]
  MoveL 131 to (300, 100, 54.07) mm, rotated rx 0.88 ry 30 rz 90.41 deg; joints [-56.114, -39.951, 132.739, -148.279, 91.611, 91.494]
  MoveL 132 to (300, 125, 54.07) mm, rotated rx 0.88 ry 30 rz 90.41 deg; joints [-57.815, -40.144, 133.987, -149.96, 92.567, 91.952]
  MoveL 133 to (300, 150, 54.09) mm, rotated rx 1.72 ry 29.81 rz 90.8 deg; joints [-59.654, -40.811, 135.395, -151.991, 92.556, 92.213]
  Set speed (1000.0 mm/s)
  MoveL 134 to (300, 150, 54.09) mm, rotated rx 1.72 ry 29.81 rz 90.8 deg; joints [-59.654, -40.811, 135.395, -151.991, 92.556, 92.213]
  MoveL 135 to (297.4, 150.32, -45.87) mm, rotated rx 1.72 ry 29.81 rz 90.8 deg; joints [-55.298, -41.624, 143.559, -147.256, 98.58, 96.486]

--- program Section2 (robot KUKA KR 5 arc) ---
  Set Ref.: Section2
  Set Tool: Paint gun
  Show Paint gun
  Set speed (1000.0 mm/s)
  MoveJ 1 to (-49.11, -1.63, 233.93) mm, rotated rx -11.88 ry 11.98 rz -21.96 deg; joints [-102.843, -5.048, 116.995, 148.178, 97.842, 8.957]
  MoveL 2 to (-49.11, -1.63, 233.93) mm, rotated rx -11.88 ry 11.98 rz -21.96 deg; joints [-102.843, -5.048, 116.995, 148.178, 97.842, 8.957]
  MoveL 3 to (0, 0, 321.03) mm, rotated rx -11.88 ry 11.98 rz -21.96 deg; joints [-101.097, -11.096, 114.649, 150.21, 90.902, 13.723]
  MoveL 4 to (0, 0, 321.03) mm, rotated rx -11.88 ry 11.98 rz -21.96 deg; joints [-101.097, -11.096, 114.649, 150.21, 90.902, 13.723]
  Set speed (20.0 mm/s)
  MoveL 5 to (0, 25, 320.56) mm, rotated rx -11.88 ry 11.98 rz -21.96 deg; joints [-99.208, -11.131, 115.208, 152.047, 91.578, 13.866]
  MoveL 6 to (0, 50, 320.21) mm, rotated rx -11.24 ry 11.1 rz -22 deg; joints [-97.197, -11.73, 116.116, 154.235, 91.144, 14.677]
  MoveL 7 to (0, 75, 319.86) mm, rotated rx -10.91 ry 11.1 rz -22.1 deg; joints [-95.139, -11.816, 116.601, 156.485, 91.67, 15.251]
  MoveL 8 to (0, 100, 319.53) mm, rotated rx -11.51 ry 10.71 rz -21.85 deg; joints [-93.448, -11.995, 116.89, 157.553, 91.656, 15.112]
  MoveL 9 to (0, 125, 319.19) mm, rotated rx -11.72 ry 12.42 rz -22.1 deg; joints [-91.278, -11.064, 116.553, 160.034, 94.098, 15.282]
  MoveL 10 to (0, 150, 318.85) mm, rotated rx -11.38 ry 10.8 rz -21.9 deg; joints [-89.428, -12.067, 117.331, 161.595, 92.427, 16.076]
  MoveL 11 to (0, 175, 318.49) mm, rotated rx -11.32 ry 11.07 rz -21.97 deg; joints [-87.371, -11.983, 117.364, 163.73, 92.952, 16.609]
  MoveL 12 to (0, 200, 318.12) mm, rotated rx -11.32 ry 11.07 rz -21.97 deg; joints [-85.378, -12.049, 117.396, 165.68, 93.059, 17.128]
  MoveL 13 to (0, 225, 317.8) mm, rotated rx -11.06 ry 10.62 rz -21.97 deg; joints [-83.369, -12.404, 117.543, 167.685, 92.506, 17.896]
  MoveL 14 to (0, 250, 317.46) mm, rotated rx -11.33 ry 10.75 rz -21.91 deg; joints [-81.466, -12.377, 117.339, 169.39, 92.602, 18.197]
  MoveL 15 to (0, 275, 317.08) mm, rotated rx -10.39 ry 9.99 rz -22.06 deg; joints [-79.287, -13.013, 117.542, 171.941, 91.357, 19.57]
  MoveL 16 to (0, 300, 316.81) mm, rotated rx -11.1 ry 10.61 rz -21.96 deg; joints [-77.489, -12.659, 116.963, 173.405, 91.92, 19.48]
  MoveL 17 to (25, 300, 304.03) mm, rotated rx -10.33 ry 9 rz -21.92 deg; joints [-77.352, -16.039, 120.619, 173.501, 90.532, 20.095]
  MoveL 18 to (25, 275, 304.3) mm, rotated rx -10.33 ry 9 rz -21.92 deg; joints [-79.332, -15.947, 120.898, 171.58, 90.834, 19.546]
  MoveL 19 to (25, 250, 304.62) mm, rotated rx -10.45 ry 8.95 rz -21.87 deg; joints [-81.389, -15.87, 121.093, 169.471, 90.99, 18.872]
  MoveL 20 to (25, 225, 304.95) mm, rotated rx -10.25 ry 9.04 rz -21.95 deg; joints [-83.309, -15.768, 121.224, 167.795, 91.163, 18.493]
  MoveL 21 to (25, 200, 305.29) mm, rotated rx -10.57 ry 8.47 rz -21.76 deg; joints [-85.549, -15.968, 121.374, 165.188, 90.493, 17.67]
  MoveL 22 to (25, 175, 305.6) mm, rotated rx -9.94 ry 8.84 rz -22.01 deg; joints [-87.279, -15.783, 121.364, 164.11, 90.774, 17.677]
  MoveL 23 to (25, 150, 305.83) mm, rotated rx -10.35 ry 8.71 rz -21.87 deg; joints [-89.477, -15.737, 121.225, 161.635, 90.46, 16.816]
  MoveL 24 to (25, 125, 306.13) mm, rotated rx -10.37 ry 8 rz -21.75 deg; joints [-91.609, -16.077, 121.226, 159.341, 89.281, 16.395]
  MoveL 25 to (25, 100, 306.51) mm, rotated rx -10.32 ry 8.46 rz -21.84 deg; joints [-93.526, -15.781, 120.862, 157.678, 89.461, 15.989]
  MoveL 26 to (25, 75, 306.8) mm, rotated rx -10.39 ry 8.89 rz -21.88 deg; joints [-95.48, -15.482, 120.408, 155.872, 89.551, 15.52]
  MoveL 27 to (25, 50, 307.11) mm, rotated rx -10.32 ry 8.91 rz -21.91 deg; joints [-97.424, -15.446, 120.022, 154.055, 89.028, 15.276]
  MoveL 28 to (25, 25, 307.4) mm, rotated rx -10.32 ry 8.91 rz -21.91 deg; joints [-99.372, -15.41, 119.55, 152.173, 88.421, 15.042]
  MoveL 29 to (25, 0, 307.67) mm, rotated rx -10.52 ry 9.29 rz -21.91 deg; joints [-101.31, -15.13, 118.853, 150.257, 88.234, 14.672]
  MoveL 30 to (50, 0, 295.9) mm, rotated rx -9.67 ry 7.17 rz -21.84 deg; joints [-101.58, -18.873, 122.401, 150.003, 85.858, 15.398]
  MoveL 31 to (50, 25, 295.67) mm, rotated rx -9.53 ry 7.93 rz -22 deg; joints [-99.487, -18.501, 122.837, 152.366, 87.52, 15.536]
  MoveL 32 to (50, 50, 295.42) mm, rotated rx -9.56 ry 7.15 rz -21.87 deg; joints [-97.627, -18.977, 123.464, 153.889, 87.113, 15.874]
  MoveL 33 to (50, 75, 295.22) mm, rotated rx -9.57 ry 6.66 rz -21.8 deg; joints [-95.698, -19.3, 123.963, 155.583, 87.005, 16.251]
  MoveL 34 to (50, 100, 294.92) mm, rotated rx -9.07 ry 6.46 rz -21.92 deg; joints [-93.535, -19.531, 124.449, 157.955, 87.181, 17.029]
  MoveL 35 to (50, 125, 294.62) mm, rotated rx -9.76 ry 6.15 rz -21.67 deg; joints [-91.794, -19.658, 124.621, 159.015, 87.209, 16.937]
  MoveL 36 to (50, 150, 294.28) mm, rotated rx -8.95 ry 5.85 rz -21.87 deg; joints [-89.509, -20.004, 125.031, 161.682, 87.039, 18.073]
  MoveL 37 to (50, 175, 294) mm, rotated rx -9.11 ry 5.67 rz -21.8 deg; joints [-87.547, -20.141, 125.136, 163.376, 87.029, 18.457]
  MoveL 38 to (50, 200, 293.84) mm, rotated rx -9.45 ry 5.95 rz -21.74 deg; joints [-85.577, -20.006, 125.033, 165.104, 87.521, 18.679]
  MoveL 39 to (50, 225, 293.54) mm, rotated rx -9.74 ry 7.08 rz -21.81 deg; joints [-83.442, -19.389, 124.671, 167.34, 89.03, 18.908]
  MoveL 40 to (50, 250, 293.21) mm, rotated rx -8.74 ry 5.41 rz -21.88 deg; joints [-81.33, -20.578, 125.085, 169.468, 86.602, 20.391]
  MoveL 41 to (50, 275, 292.97) mm, rotated rx -8.65 ry 5.28 rz -21.89 deg; joints [-79.3, -20.751, 124.911, 171.418, 86.205, 21.016]
  MoveL 42 to (50, 300, 292.68) mm, rotated rx -9 ry 5.29 rz -21.79 deg; joints [-77.424, -20.78, 124.584, 172.96, 86, 21.266]
  MoveL 43 to (75, 300, 282.71) mm, rotated rx -8.17 ry 3.91 rz -21.87 deg; joints [-77.277, -24.245, 127.556, 173.134, 84.041, 22.017]
  MoveL 44 to (75, 275, 282.93) mm, rotated rx -8.07 ry 3.66 rz -21.87 deg; joints [-79.311, -24.318, 127.915, 171.181, 84.002, 21.591]
  MoveL 45 to (75, 250, 283.17) mm, rotated rx -8.05 ry 3.75 rz -21.88 deg; joints [-81.327, -24.184, 128.12, 169.33, 84.334, 21.07]
  MoveL 46 to (75, 225, 283.42) mm, rotated rx -8.26 ry 3.89 rz -21.84 deg; joints [-83.438, -23.985, 128.204, 167.24, 84.688, 20.353]
  MoveL 47 to (75, 200, 283.63) mm, rotated rx -8.22 ry 3.8 rz -21.84 deg; joints [-85.507, -23.966, 128.289, 165.276, 84.573, 19.862]
  MoveL 48 to (75, 175, 283.93) mm, rotated rx -8.33 ry 4.07 rz -21.84 deg; joints [-87.574, -23.721, 128.201, 163.347, 84.862, 19.234]
  MoveL 49 to (75, 150, 284.16) mm, rotated rx -8.34 ry 4.03 rz -21.83 deg; joints [-89.659, -23.674, 128.107, 161.346, 84.628, 18.74]
  MoveL 50 to (75, 125, 284.38) mm, rotated rx -8.5 ry 3.92 rz -21.77 deg; joints [-91.797, -23.654, 127.92, 159.166, 84.213, 18.194]
  MoveL 51 to (75, 100, 284.62) mm, rotated rx -8.16 ry 3.98 rz -21.88 deg; joints [-93.722, -23.62, 127.726, 157.603, 83.882, 18.041]
  MoveL 52 to (75, 75, 284.9) mm, rotated rx -8.48 ry 3.79 rz -21.76 deg; joints [-95.894, -23.623, 127.347, 155.242, 83.207, 17.51]
  MoveL 53 to (75, 50, 285.03) mm, rotated rx -7.97 ry 4.22 rz -21.96 deg; joints [-97.679, -23.411, 127.007, 154.056, 83.224, 17.501]
  MoveL 54 to (75, 25, 285.28) mm, rotated rx -9.03 ry 4.64 rz -21.7 deg; joints [-99.978, -22.96, 126.193, 151.213, 83.243, 16.444]
  MoveL 55 to (75, 0, 285.59) mm, rotated rx -8.29 ry 4.92 rz -21.95 deg; joints [-101.658, -22.872, 125.78, 150.228, 82.916, 16.757]
  MoveL 56 to (100, 0, 276.46) mm, rotated rx -7.31 ry 2.55 rz -21.97 deg; joints [-101.853, -26.978, 128.723, 149.9, 79.452, 18.098]
  MoveL 57 to (100, 25, 276.18) mm, rotated rx -8.01 ry 2.3 rz -21.74 deg; joints [-100.136, -27.062, 129.147, 150.968, 79.815, 17.828]
  MoveL 58 to (100, 50, 275.97) mm, rotated rx -7.3 ry 1.38 rz -21.86 deg; joints [-98.007, -27.77, 129.893, 153.174, 79.043, 18.739]
  MoveL 59 to (100, 75, 275.79) mm, rotated rx -7.63 ry 2.62 rz -21.88 deg; joints [-95.927, -27.06, 130.116, 155.392, 81.319, 18.428]
  MoveL 60 to (100, 100, 275.62) mm, rotated rx -7.34 ry 0.98 rz -21.81 deg; joints [-94, -28.11, 130.667, 156.802, 79.436, 19.35]
  MoveL 61 to (100, 125, 275.44) mm, rotated rx -7.44 ry 2.24 rz -21.9 deg; joints [-91.781, -27.43, 130.78, 159.321, 81.561, 19.35]
  MoveL 62 to (100, 150, 275.23) mm, rotated rx -7.56 ry 2.16 rz -21.86 deg; joints [-89.752, -27.52, 130.941, 161.116, 81.739, 19.698]
  MoveL 63 to (100, 175, 275.02) mm, rotated rx -7.58 ry 2.22 rz -21.85 deg; joints [-87.661, -27.551, 131.026, 163.09, 82, 20.128]
  MoveL 64 to (100, 200, 274.81) mm, rotated rx -7.61 ry 2.28 rz -21.85 deg; joints [-85.566, -27.585, 131.031, 165.067, 82.166, 20.59]
  MoveL 65 to (100, 225, 274.59) mm, rotated rx -7.61 ry 2.28 rz -21.85 deg; joints [-83.478, -27.663, 130.967, 167.029, 82.145, 21.097]
  MoveL 66 to (100, 250, 274.37) mm, rotated rx -7.53 ry 1.74 rz -21.82 deg; joints [-81.469, -28.066, 130.905, 168.753, 81.272, 21.74]
  MoveL 67 to (100, 275, 274.18) mm, rotated rx -7.14 ry 0.88 rz -21.86 deg; joints [-79.427, -28.713, 130.835, 170.58, 79.754, 22.645]
  MoveL 68 to (100, 300, 273.98) mm, rotated rx -7.2 ry 1.68 rz -21.91 deg; joints [-77.261, -28.327, 130.414, 172.906, 80.533, 22.989]
  MoveL 69 to (125, 300, 266.45) mm, rotated rx -6.38 ry -0.19 rz -21.98 deg; joints [-77.259, -32.288, 132.882, 172.65, 77.129, 23.886]
  MoveL 70 to (125, 275, 267.13) mm, rotated rx 5.94 ry -26.96 rz -26.11 deg; joints [-80.82, -45.444, 129.768, 155.408, 34.805, 44.696]
  MoveL 71 to (125, 250, 266.79) mm, rotated rx -6.68 ry -0.2 rz -21.9 deg; joints [-81.494, -32.089, 133.411, 168.482, 77.782, 22.773]
  MoveL 72 to (125, 225, 266.95) mm, rotated rx -6.23 ry -0.41 rz -22.01 deg; joints [-83.458, -32.217, 133.635, 166.869, 77.49, 22.656]
  MoveL 73 to (125, 200, 267.22) mm, rotated rx -6.76 ry 0.09 rz -21.9 deg; joints [-85.662, -31.753, 133.591, 164.655, 78.379, 21.735]
  MoveL 74 to (125, 175, 267.35) mm, rotated rx -6.09 ry 0.33 rz -22.11 deg; joints [-87.484, -31.662, 133.667, 163.522, 78.5, 21.7]
  MoveL 75 to (125, 150, 267.45) mm, rotated rx -6.59 ry 0.96 rz -22.02 deg; joints [-89.674, -31.126, 133.459, 161.372, 79.376, 20.783]
  MoveL 76 to (125, 125, 267.62) mm, rotated rx -6.3 ry -1.09 rz -21.94 deg; joints [-91.977, -32.295, 133.458, 158.554, 76.146, 21.141]
  MoveL 77 to (125, 100, 267.82) mm, rotated rx -6.57 ry 0.26 rz -21.97 deg; joints [-93.96, -31.397, 133.083, 157.061, 77.8, 20.252]
  MoveL 78 to (125, 75, 267.97) mm, rotated rx -6.4 ry -0.58 rz -21.95 deg; joints [-96.083, -31.841, 132.819, 154.804, 76.156, 20.35]
  MoveL 79 to (125, 50, 268.14) mm, rotated rx -6.4 ry -0.58 rz -21.95 deg; joints [-98.124, -31.766, 132.396, 152.847, 75.676, 20.154]
  MoveL 80 to (125, 25, 268.41) mm, rotated rx -7.09 ry 0.31 rz -21.82 deg; joints [-100.264, -31.057, 131.695, 150.664, 76.483, 19.286]
  MoveL 81 to (125, 0, 268.58) mm, rotated rx -6.69 ry 0.31 rz -21.93 deg; joints [-102.119, -31.056, 131.211, 149.135, 75.805, 19.47]
  MoveL 82 to (150, 0, 261.88) mm, rotated rx -6.18 ry -2.02 rz -21.91 deg; joints [-102.394, -35.233, 133.32, 148.046, 71.736, 21.154]
  MoveL 83 to (150, 25, 261.77) mm, rotated rx -6.13 ry -2.33 rz -21.9 deg; joints [-100.421, -35.522, 133.918, 149.882, 71.844, 21.32]
  MoveL 84 to (150, 50, 261.49) mm, rotated rx -5.71 ry -2.2 rz -22.03 deg; joints [-98.252, -35.632, 134.536, 152.36, 72.467, 21.558]
  MoveL 85 to (150, 75, 261.35) mm, rotated rx -6.04 ry -2.92 rz -21.89 deg; joints [-96.401, -36.059, 134.886, 153.575, 71.945, 21.806]
  MoveL 86 to (150, 100, 261.21) mm, rotated rx -5.44 ry -3 rz -22.06 deg; joints [-94.141, -36.313, 135.347, 156.125, 72.061, 22.374]
  MoveL 87 to (150, 125, 261.07) mm, rotated rx -5.43 ry -2.88 rz -22.06 deg; joints [-92.036, -36.331, 135.612, 158.188, 72.53, 22.58]
  MoveL 88 to (150, 150, 260.93) mm, rotated rx -5.64 ry -2.85 rz -22.01 deg; joints [-90.005, -36.357, 135.758, 159.978, 72.835, 22.745]
  MoveL 89 to (150, 175, 260.81) mm, rotated rx -5.27 ry -2.43 rz -22.14 deg; joints [-87.701, -36.268, 135.899, 162.598, 73.467, 23.176]
  MoveL 90 to (150, 200, 260.66) mm, rotated rx -5.98 ry -2.63 rz -21.92 deg; joints [-85.878, -36.321, 135.817, 163.718, 73.419, 23.171]
  MoveL 91 to (175, 175, 255.42) mm, rotated rx -4.54 ry -5.12 rz -22.2 deg; joints [-87.938, -40.877, 137.686, 161.386, 68.137, 24.911]
  MoveL 92 to (175, 150, 255.55) mm, rotated rx -3.65 ry -5.36 rz -22.44 deg; joints [-89.775, -41.116, 137.694, 160.116, 67.375, 25.234]
  MoveL 93 to (175, 125, 255.73) mm, rotated rx -4.92 ry -4.62 rz -22.12 deg; joints [-92.205, -40.351, 137.383, 157.327, 68.714, 24.026]
  MoveL 94 to (175, 100, 255.75) mm, rotated rx -4.63 ry -4.72 rz -22.19 deg; joints [-94.21, -40.364, 137.167, 155.55, 68.246, 24.042]
  MoveL 95 to (175, 75, 255.88) mm, rotated rx -4.59 ry -4.74 rz -22.2 deg; joints [-96.272, -40.278, 136.823, 153.563, 67.879, 23.951]
  MoveL 96 to (175, 50, 255.98) mm, rotated rx -4.65 ry -4.72 rz -22.19 deg; joints [-98.337, -40.139, 136.382, 151.506, 67.536, 23.853]
  MoveL 97 to (175, 25, 256.14) mm, rotated rx -4.79 ry -4.17 rz -22.17 deg; joints [-100.346, -39.689, 135.878, 149.726, 67.922, 23.5]
  MoveL 98 to (175, 0, 256.25) mm, rotated rx -5 ry -4.3 rz -22.11 deg; joints [-102.421, -39.575, 135.219, 147.408, 67.284, 23.538]
  MoveL 99 to (200, 0, 251.75) mm, rotated rx -4.17 ry -6.29 rz -22.26 deg; joints [-102.502, -43.72, 136.689, 146.295, 63.015, 25.973]
  MoveL 100 to (200, 25, 251.71) mm, rotated rx -4.08 ry -6.17 rz -22.29 deg; joints [-100.47, -43.85, 137.33, 148.54, 63.594, 25.775]
  MoveL 101 to (200, 50, 251.58) mm, rotated rx -3.44 ry -7.61 rz -22.43 deg; joints [-98.397, -44.877, 137.767, 150.12, 61.673, 26.87]
  MoveL 102 to (200, 75, 251.51) mm, rotated rx -3.19 ry -7.13 rz -22.51 deg; joints [-96.216, -44.841, 138.314, 152.815, 62.59, 26.639]
  MoveL 103 to (200, 100, 251.56) mm, rotated rx -4 ry -7.15 rz -22.28 deg; joints [-94.419, -44.799, 138.525, 154.032, 63.093, 26.31]
  MoveL 104 to (200, 125, 251.39) mm, rotated rx -4.19 ry -6.62 rz -22.24 deg; joints [-92.328, -44.599, 138.842, 156.293, 64.15, 25.995]
  MoveL 105 to (200, 150, 251.31) mm, rotated rx -3.81 ry -6.98 rz -22.34 deg; joints [-90.152, -44.971, 139.029, 158.441, 63.61, 26.485]
  MoveL 106 to (225, 150, 248.03) mm, rotated rx -2.53 ry -9.87 rz -22.65 deg; joints [-90.227, -49.767, 139.988, 156.84, 57.128, 29.529]
  MoveL 107 to (225, 125, 248.12) mm, rotated rx -2.35 ry -9.2 rz -22.7 deg; joints [-92.154, -49.375, 139.957, 155.543, 57.974, 29.164]
  MoveL 108 to (225, 100, 248.17) mm, rotated rx -2.65 ry -9.1 rz -22.62 deg; joints [-94.321, -49.123, 139.678, 153.222, 58.129, 29.019]
  MoveL 109 to (225, 75, 248.22) mm, rotated rx -2.69 ry -9.01 rz -22.61 deg; joints [-96.385, -48.918, 139.338, 151.153, 58.093, 29.03]
  MoveL 110 to (225, 50, 248.27) mm, rotated rx -2.72 ry -9.07 rz -22.6 deg; joints [-98.44, -48.766, 138.881, 148.951, 57.778, 29.213]
  MoveL 111 to (225, 25, 248.29) mm, rotated rx -2.63 ry -9 rz -22.63 deg; joints [-100.416, -48.559, 138.388, 146.987, 57.571, 29.397]
  MoveL 112 to (225, 0, 248.34) mm, rotated rx -2.74 ry -9.11 rz -22.59 deg; joints [-102.441, -48.365, 137.733, 144.642, 57.137, 29.723]
  MoveL 113 to (250, 0, 246.02) mm, rotated rx -1.64 ry -11.38 rz -22.89 deg; joints [-102.41, -52.562, 138.366, 142.461, 51.971, 33.582]
  MoveL 114 to (250, 25, 245.99) mm, rotated rx -1.6 ry -10.83 rz -22.9 deg; joints [-100.376, -52.615, 139.133, 145.315, 52.901, 32.674]
  MoveL 115 to (250, 50, 246.08) mm, rotated rx -1.6 ry -10.83 rz -22.9 deg; joints [-98.369, -52.843, 139.647, 147.511, 53.075, 32.354]
  MoveL 116 to (250, 75, 246.1) mm, rotated rx -0.18 ry -11.17 rz -23.28 deg; joints [-95.917, -53.526, 140.16, 150.789, 52.052, 32.824]
  MoveL 117 to (250, 100, 245.97) mm, rotated rx -1.11 ry -12.04 rz -23.04 deg; joints [-94.282, -53.84, 140.184, 151.085, 51.375, 33.059]
  MoveL 118 to (250, 125, 245.94) mm, rotated rx -1.8 ry -12.48 rz -22.86 deg; joints [-92.509, -54.016, 140.263, 152.074, 51.124, 33.033]
  MoveL 119 to (250, 150, 245.94) mm, rotated rx -1.11 ry -12 rz -23.04 deg; joints [-90.144, -54.105, 140.622, 155.492, 51.446, 32.646]
  MoveL 120 to (275, 150, 244.77) mm, rotated rx -0.36 ry -13.41 rz -23.27 deg; joints [-90.178, -57.872, 141.011, 153.689, 46.953, 35.461]
  MoveL 121 to (275, 125, 244.75) mm, rotated rx -0.5 ry -13.98 rz -23.25 deg; joints [-92.368, -57.906, 140.661, 150.539, 46.343, 36.347]
  MoveL 122 to (275, 100, 244.83) mm, rotated rx -0.72 ry -13.98 rz -23.19 deg; joints [-94.48, -57.68, 140.371, 148.031, 46.51, 36.671]
  MoveL 123 to (275, 75, 244.77) mm, rotated rx -0.67 ry -13.02 rz -23.18 deg; joints [-96.379, -57.149, 140.331, 147.043, 47.794, 36.018]
  MoveL 124 to (275, 50, 244.76) mm, rotated rx -0.66 ry -13.72 rz -23.2 deg; joints [-98.466, -57.157, 139.673, 143.854, 46.838, 37.238]
  MoveL 125 to (275, 25, 244.79) mm, rotated rx -0.66 ry -13.72 rz -23.2 deg; joints [-100.446, -56.882, 139.14, 141.548, 46.791, 37.739]
  MoveL 126 to (275, 0, 244.79) mm, rotated rx -0.91 ry -13.15 rz -23.12 deg; joints [-102.426, -56.326, 138.676, 139.753, 47.576, 37.541]
  MoveL 127 to (300, 0, 244.61) mm, rotated rx 0.12 ry -15.38 rz -23.46 deg; joints [-102.367, -60.105, 138.487, 135.807, 42.507, 43.032]
  MoveL 128 to (300, 25, 244.59) mm, rotated rx 0.12 ry -15.38 rz -23.46 deg; joints [-100.43, -60.452, 139.106, 138.215, 42.443, 42.34]
  MoveL 129 to (300, 50, 244.6) mm, rotated rx 0.46 ry -15.86 rz -23.58 deg; joints [-98.408, -60.972, 139.489, 140.194, 41.58, 42.448]
  MoveL 130 to (300, 75, 244.63) mm, rotated rx 0.46 ry -15.86 rz -23.58 deg; joints [-96.42, -61.241, 139.926, 142.608, 41.465, 41.827]
  MoveL 131 to (300, 100, 244.66) mm, rotated rx 0.46 ry -15.86 rz -23.58 deg; joints [-94.41, -61.47, 140.273, 145.017, 41.329, 41.243]
  MoveL 132 to (300, 125, 244.7) mm, rotated rx 0.31 ry -15.3 rz -23.51 deg; joints [-92.356, -61.463, 140.72, 148.122, 41.975, 39.925]
  MoveL 133 to (300, 150, 244.77) mm, rotated rx 0.31 ry -15.12 rz -23.51 deg; joints [-90.282, -61.556, 140.945, 150.787, 42.029, 39.194]
  Set speed (1000.0 mm/s)
  MoveL 134 to (300, 150, 244.77) mm, rotated rx 0.31 ry -15.12 rz -23.51 deg; joints [-90.282, -61.556, 140.945, 150.787, 42.029, 39.194]
  MoveL 135 to (300.4, 150.4, 144.77) mm, rotated rx 0.31 ry -15.12 rz -23.51 deg; joints [-90.662, -65.515, 150.914, 153.218, 47.362, 35.247]

--- program MainInspection Part (robot KUKA KR 5 arc) ---
  Call Section1
  Call Section2
